

FUNCTION FC31 : VOID //FC de rearranjo para envio ao CLP de Elétrica
VAR
    tmp1: DINT;
    tmp2: DINT;
    tmp3: DINT;
END_VAR


BEGIN //code section




   QW46 := DINT_TO_WORD((tmp1 + tmp2 + tmp3 )/3);//  Analógicas - Média entre fases -  M-B-512401B










END_FUNCTION